# EPICS autosave request: luaApp/Db/luascripts10_settings.req
file script_settings.req P=$(P)$(R)userScript1
file script_settings.req P=$(P)$(R)userScript2
file script_settings.req P=$(P)$(R)userScript3
file script_settings.req P=$(P)$(R)userScript4
file script_settings.req P=$(P)$(R)userScript5
file script_settings.req P=$(P)$(R)userScript6
file script_settings.req P=$(P)$(R)userScript7
file script_settings.req P=$(P)$(R)userScript8
file script_settings.req P=$(P)$(R)userScript9
file script_settings.req P=$(P)$(R)userScript0
